FUNCTION_BLOCK UA_SkillIds (* OPC UA node IDs of one skill facade, below UaRoot *)
  (* Standard: 61499-2 *)
  (* Version 2.0, 2026-09-27, Project contributors, Filling cell reference model *)
  PACKAGE fillingcell;
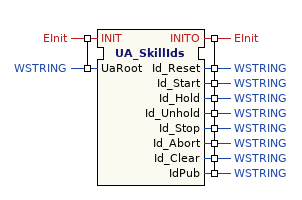
  EVENT_INPUT
    INIT : EInit WITH UaRoot;
  END_EVENT
  EVENT_OUTPUT
    INITO : EInit WITH Id_Reset, Id_Start, Id_Hold, Id_Unhold, Id_Stop, Id_Abort, Id_Clear, IdPub;
  END_EVENT
  VAR_INPUT
    UaRoot : WSTRING;
  END_VAR
  VAR_OUTPUT
    Id_Reset : WSTRING;
    Id_Start : WSTRING;
    Id_Hold : WSTRING;
    Id_Unhold : WSTRING;
    Id_Stop : WSTRING;
    Id_Abort : WSTRING;
    Id_Clear : WSTRING;
    IdPub : WSTRING;
  END_VAR
  EC_STATES
    INIT : INIT -> INITO;
  END_STATES
  ALGORITHM INIT IN ST:
Id_Reset := CONCAT(CONCAT("opc_ua[CREATE_METHOD;", UaRoot), "/Reset]");
Id_Start := CONCAT(CONCAT("opc_ua[CREATE_METHOD;", UaRoot), "/Start]");
Id_Hold := CONCAT(CONCAT("opc_ua[CREATE_METHOD;", UaRoot), "/Hold]");
Id_Unhold := CONCAT(CONCAT("opc_ua[CREATE_METHOD;", UaRoot), "/Unhold]");
Id_Stop := CONCAT(CONCAT("opc_ua[CREATE_METHOD;", UaRoot), "/Stop]");
Id_Abort := CONCAT(CONCAT("opc_ua[CREATE_METHOD;", UaRoot), "/Abort]");
Id_Clear := CONCAT(CONCAT("opc_ua[CREATE_METHOD;", UaRoot), "/Clear]");
IdPub := CONCAT(CONCAT(CONCAT(CONCAT(CONCAT(CONCAT(CONCAT(CONCAT(CONCAT(CONCAT(CONCAT(CONCAT("opc_ua[WRITE;", UaRoot), "/State;"), UaRoot), "/ErrorID;"), UaRoot), "/P1;"), UaRoot), "/P2;"), UaRoot), "/P3;"), UaRoot), "/P4]");
  END_ALGORITHM
END_FUNCTION_BLOCK
